(* IEC 61131-3 sources: SmartHomeNew/ (part 17) *)

(* ---- PRG_Telemetry_Causality_Governor.st ---- *)
PROGRAM PRG_Telemetry_Causality_Governor
VAR
    L_Now_MS : UDINT;
    L_Causality_Valid : BOOL := TRUE;
    L_Error_Code : UDINT := 0;
    L_Error_Text : STRING(160) := '';
    L_Ack_Age_MS : UDINT;
    L_Convergence_Age_MS : UDINT;
    L_Stable_Dwell_MS : UDINT;
END_VAR

L_Now_MS := GVL_STATUS.G_System_Time_MS;
L_Causality_Valid := TRUE;
L_Error_Code := 0;
L_Error_Text := '';

// Fail-safe defaults.
GVL_TELEMETRY.Telemetry_Runtime_Valid := FALSE;
GVL_TELEMETRY.Telemetry_Freshness_Valid := FALSE;
GVL_TELEMETRY.Command_Telemetry_Causality_Valid := FALSE;
GVL_TELEMETRY.Actuator_Feedback_Valid := FALSE;
GVL_TELEMETRY.Actuator_Feedback_Fresh := FALSE;
GVL_TELEMETRY.Physical_Effect_Confirmed := FALSE;
GVL_TELEMETRY.Physical_Effect_Finalized := FALSE;
GVL_TELEMETRY.Physical_Target_Converged := FALSE;
GVL_TELEMETRY.Physical_Stable_Window_OK := FALSE;
GVL_TELEMETRY.Command_Telemetry_Divergence_Detected := TRUE;

GVL_TELEMETRY.Command_Epoch := GVL_OUTPUT_EPOCH.Output_Publication_Epoch;

IF NOT GVL_OUTPUT_EPOCH.Output_Publication_Valid THEN
    L_Causality_Valid := FALSE;
    L_Error_Code := 21000;
    L_Error_Text := 'Telemetry causality output publication invalid';
END_IF;

IF L_Causality_Valid AND NOT GVL_OUTPUT_EPOCH.Output_Runtime_Epoch_Valid THEN
    L_Causality_Valid := FALSE;
    L_Error_Code := 21001;
    L_Error_Text := 'Telemetry causality runtime epoch invalid';
END_IF;

IF L_Causality_Valid AND GVL_OUTPUT_EPOCH.Output_Lease_Expired THEN
    L_Causality_Valid := FALSE;
    L_Error_Code := 21002;
    L_Error_Text := 'Telemetry causality output lease expired';
END_IF;

IF L_Causality_Valid AND GVL_OUTPUT_EPOCH.Output_Forced_Safe_Decay THEN
    L_Causality_Valid := FALSE;
    L_Error_Code := 21003;
    L_Error_Text := 'Telemetry causality output forced safe decay';
END_IF;

IF L_Causality_Valid AND (GVL_TELEMETRY.Telemetry_Epoch <> GVL_TELEMETRY.Command_Epoch) THEN
    L_Causality_Valid := FALSE;
    L_Error_Code := 21010;
    L_Error_Text := 'Telemetry epoch does not match command epoch';
END_IF;

IF L_Causality_Valid AND (GVL_TELEMETRY.Telemetry_Epoch < GVL_TELEMETRY.Last_Acknowledged_Command_Epoch) THEN
    GVL_TELEMETRY.Telemetry_Replay_Suspected := TRUE;

    L_Causality_Valid := FALSE;
    L_Error_Code := 21011;
    L_Error_Text := 'Telemetry epoch replay suspected';
END_IF;

L_Ack_Age_MS := L_Now_MS - GVL_TELEMETRY.Last_Physical_Ack_Time_MS;

IF L_Causality_Valid AND (L_Ack_Age_MS > 5000) THEN
    L_Causality_Valid := FALSE;
    L_Error_Code := 21020;
    L_Error_Text := 'Physical acknowledgement stale';
END_IF;

L_Convergence_Age_MS := L_Now_MS - GVL_TELEMETRY.Last_Physical_Convergence_MS;

IF L_Causality_Valid AND (L_Convergence_Age_MS > 10000) THEN
    L_Causality_Valid := FALSE;
    L_Error_Code := 21021;
    L_Error_Text := 'Physical convergence stale';
END_IF;

// Stable physical dwell window.
L_Stable_Dwell_MS :=
    L_Now_MS - GVL_TELEMETRY.Last_Physical_Convergence_MS;

IF L_Causality_Valid AND (L_Stable_Dwell_MS < 3000) THEN
    L_Causality_Valid := FALSE;
    L_Error_Code := 21030;
    L_Error_Text := 'Physical stabilization dwell window incomplete';
END_IF;

// Physical oscillation quarantine.
IF L_Causality_Valid
AND GVL_TELEMETRY.Physical_Oscillation_Detected THEN
    L_Causality_Valid := FALSE;
    L_Error_Code := 21031;
    L_Error_Text := 'Physical oscillation detected';
END_IF;

IF L_Causality_Valid
AND GVL_TELEMETRY.Physical_Transition_Active THEN
    L_Causality_Valid := FALSE;
    L_Error_Code := 21032;
    L_Error_Text := 'Physical transition still active';
END_IF;

IF L_Causality_Valid
AND GVL_TELEMETRY.Physical_Convergence_Replay_Suspected THEN
    L_Causality_Valid := FALSE;
    L_Error_Code := 21033;
    L_Error_Text := 'Physical convergence replay suspected';
END_IF;

IF L_Causality_Valid THEN
    GVL_TELEMETRY.Telemetry_Runtime_Valid := TRUE;
    GVL_TELEMETRY.Telemetry_Freshness_Valid := TRUE;
    GVL_TELEMETRY.Telemetry_Lease_Expired := FALSE;
    GVL_TELEMETRY.Telemetry_Quarantine_Active := FALSE;

    GVL_TELEMETRY.Command_Telemetry_Causality_Valid := TRUE;
    GVL_TELEMETRY.Command_Telemetry_Divergence_Detected := FALSE;

    GVL_TELEMETRY.Actuator_Feedback_Valid := TRUE;
    GVL_TELEMETRY.Actuator_Feedback_Fresh := TRUE;
    GVL_TELEMETRY.Physical_Effect_Confirmed := TRUE;

    GVL_TELEMETRY.Physical_Target_Converged := TRUE;
    GVL_TELEMETRY.Physical_Stable_Window_OK := TRUE;
    GVL_TELEMETRY.Physical_Effect_Finalized := TRUE;

    GVL_TELEMETRY.Last_Acknowledged_Command_Epoch := GVL_TELEMETRY.Command_Epoch;

    GVL_TELEMETRY.Telemetry_Last_Error_Code := 0;
    GVL_TELEMETRY.Telemetry_Last_Error_Text := '';
ELSE
    GVL_TELEMETRY.Telemetry_Runtime_Valid := FALSE;
    GVL_TELEMETRY.Telemetry_Freshness_Valid := FALSE;
    GVL_TELEMETRY.Telemetry_Lease_Expired := TRUE;
    GVL_TELEMETRY.Telemetry_Quarantine_Active := TRUE;

    GVL_TELEMETRY.Command_Telemetry_Causality_Valid := FALSE;
    GVL_TELEMETRY.Command_Telemetry_Divergence_Detected := TRUE;

    GVL_TELEMETRY.Telemetry_Last_Error_Code := L_Error_Code;
    GVL_TELEMETRY.Telemetry_Last_Error_Text := L_Error_Text;
    GVL_TELEMETRY.Telemetry_Invalidation_Count :=
        GVL_TELEMETRY.Telemetry_Invalidation_Count + 1;
END_IF;

END_PROGRAM

(* ---- PRG_Temporal_Domain.st ---- *)
PROGRAM PRG_Temporal_Domain
// SEMANTIC DOMAIN WRAPPER
// PRESERVES ORIGINAL EXECUTION ORDER

PRG_Temporal_Stability_Governor();
PRG_Control_Temporal_Coherence_Governor();

PRG_Temporal_Causality_Closure_Governor();
PRG_Distributed_Epoch_Linearity_Governor();
PRG_Historical_Ordering_Integrity_Governor();
PRG_Causality_Reversal_Prevention_Governor();

END_PROGRAM

(* ---- PRG_Test.st ---- *)
PROGRAM PRG_Test
VAR
    // Инстансы тестируемых блоков
    fbAnalogValidator : FB_Analog_Validator;
    fbRandomGenerator : FB_Random_Generator;
    fbTwoFactorAuth   : FB_TwoFactor_Auth;

    // Переменные для тестов
    L_Test_Step : INT := 0;
    L_Tests_Passed : INT := 0;
    L_Tests_Failed : INT := 0;
    L_System_Time : UDINT := 0;

    // Результаты тестов
    L_Test1_Passed : BOOL;
    L_Test2_Passed : BOOL;
    L_Test3_Passed : BOOL;
END_VAR

// Имитация системного времени
L_System_Time := L_System_Time + 10;

CASE L_Test_Step OF
    0: // Инициализация
        L_Test_Step := 1;

    1: // Тест 1: FB_Analog_Validator - Нормальное значение
        fbAnalogValidator(
            VI_Value := 25.0,
            VI_Min_Valid := 0.0,
            VI_Max_Valid := 50.0,
            VI_Fallback_Mode := 0,
            VI_Default_Value := 20.0
        );
        IF fbAnalogValidator.VO_Valid AND fbAnalogValidator.VO_Validated_Value = 25.0 THEN
            L_Test1_Passed := TRUE;
            L_Tests_Passed := L_Tests_Passed + 1;
        ELSE
            L_Test1_Passed := FALSE;
            L_Tests_Failed := L_Tests_Failed + 1;
        END_IF;
        L_Test_Step := 2;

    2: // Тест 2: FB_Analog_Validator - Выход за границы (Fallback = Default)
        fbAnalogValidator(
            VI_Value := 100.0,
            VI_Min_Valid := 0.0,
            VI_Max_Valid := 50.0,
            VI_Fallback_Mode := 1,
            VI_Default_Value := 20.0
        );
        IF NOT fbAnalogValidator.VO_Valid AND fbAnalogValidator.VO_Validated_Value = 20.0 THEN
            L_Test2_Passed := TRUE;
            L_Tests_Passed := L_Tests_Passed + 1;
        ELSE
            L_Test2_Passed := FALSE;
            L_Tests_Failed := L_Tests_Failed + 1;
        END_IF;
        L_Test_Step := 3;

    3: // Тест 3: FB_Random_Generator - Диапазон
        fbRandomGenerator.Seed(12345);
        fbRandomGenerator.Random_Int_Range(VI_min := 10, VI_max := 20, VI_System_Time_MS := L_System_Time);
        IF fbRandomGenerator.VO_Random_Value >= 10 AND fbRandomGenerator.VO_Random_Value <= 20 THEN
            L_Test3_Passed := TRUE;
            L_Tests_Passed := L_Tests_Passed + 1;
        ELSE
            L_Test3_Passed := FALSE;
            L_Tests_Failed := L_Tests_Failed + 1;
        END_IF;
        L_Test_Step := 100; // Завершение тестов

    100: // Тесты завершены
        // Здесь можно вывести результаты в лог или HMI
        ;
END_CASE;
// >>> BULK_SYNC_ANCHOR: PRG_Test <<<

(* ---- PRG_Test_Scenario_Runner.st ---- *)
PROGRAM PRG_Test_Scenario_Runner

IF NOT GVL_TEST.G_Test_Enable THEN
    RETURN;
END_IF;

CASE GVL_TEST_INJECTION.G_Test_Step OF

0:
    // idle

1:
    // simulate gas spike
    GVL_TEST_INJECTION.G_Inject_Gas_Level := 50.0;
    GVL_TEST_INJECTION.G_Test_Step := 2;

2:
    // simulate illegal reset
    GVL_TEST_INJECTION.G_Inject_Force_Gas_Alarm_Reset := TRUE;
    GVL_TEST_INJECTION.G_Test_Step := 3;

3:
    // simulate IO offline
    GVL_TEST_INJECTION.G_Inject_Force_IO_Offline := TRUE;
    GVL_TEST_INJECTION.G_Test_Step := 4;

4:
    // stop
    GVL_TEST_INJECTION.G_Inject_Enable := FALSE;

END_CASE;

(* ---- PRG_Time_Service.st ---- *)
PROGRAM PRG_Time_Service
VAR
    fbTimebase : FB_System_Timebase;
    fbTime : FB_Time_Service;
END_VAR

// Central time update point.
// Must run before PRG_IO_Read and all consumers of GVL_TIME_SERVICE.
fbTimebase();
fbTime();

// Step 4.2 compatibility bridge.
// Legacy consumers of GVL_STATUS.G_System_Time_MS receive the same canonical time.
GVL_STATUS.G_System_Time_MS := GVL_TIME_SERVICE.G_Now_MS;
GVL_STATUS.G_Current_TOD := GVL_TIME_SERVICE.G_Current_TOD;
GVL_STATUS.G_Current_Day := GVL_TIME_SERVICE.G_Day_Of_Week;

END_PROGRAM

(* ---- PRG_Transport_Freshness_Governor.st ---- *)
PROGRAM PRG_Transport_Freshness_Governor
VAR
    L_Now_MS : UDINT;
    L_Delta_MS : UDINT;
    L_Transport_Valid : BOOL := TRUE;
    L_Error_Code : UDINT := 0;
    L_Error_Text : STRING(160) := '';
END_VAR

L_Now_MS := GVL_STATUS.G_System_Time_MS;
L_Transport_Valid := TRUE;
L_Error_Code := 0;
L_Error_Text := '';

// ======================================================
// TRANSPORT FRESHNESS GOVERNOR
// ======================================================
// Governs transport freshness semantics.
// Prevents stale transport semantic publication.
// ======================================================

GVL_TRANSPORT_FRESHNESS.Transport_Stale_Frame_Detected := FALSE;
GVL_TRANSPORT_FRESHNESS.Transport_Transaction_Mismatch := FALSE;
GVL_TRANSPORT_FRESHNESS.Transport_Snapshot_Invalid := FALSE;

// Runtime authority linkage.
IF NOT GVL_RUNTIME_EPOCH.Runtime_Runtime_Barrier_OK THEN
    L_Transport_Valid := FALSE;
    L_Error_Code := 10000;
    L_Error_Text := 'Transport runtime authority invalid';
END_IF;

// Monotonic authority linkage.
IF L_Transport_Valid AND (NOT GVL_TIME_MONOTONIC.Monotonic_Time_Valid) THEN
    L_Transport_Valid := FALSE;
    L_Error_Code := 10001;
    L_Error_Text := 'Transport monotonic authority invalid';
END_IF;

// Recovery governance linkage.
IF L_Transport_Valid AND GVL_RECOVERY_GOVERNANCE.Recovery_Quarantine_Active THEN
    L_Transport_Valid := FALSE;
    L_Error_Code := 10002;
    L_Error_Text := 'Transport blocked by recovery quarantine';
END_IF;

// Transport reconnect quarantine.
IF GVL_TRANSPORT_FRESHNESS.Transport_Reconnect_Stabilizing THEN
    GVL_TRANSPORT_FRESHNESS.Transport_Quarantine_Active := TRUE;

    L_Transport_Valid := FALSE;

    IF L_Error_Code = 0 THEN
        L_Error_Code := 10003;
        L_Error_Text := 'Transport reconnect stabilization active';
    END_IF;
END_IF;

// Lease freshness validation.
L_Delta_MS := L_Now_MS - GVL_TRANSPORT_FRESHNESS.Transport_Last_Refresh_MS;

IF L_Transport_Valid AND GVL_TRANSPORT_FRESHNESS.Transport_Lease_Valid THEN
    IF L_Delta_MS > GVL_TRANSPORT_FRESHNESS.Transport_Lease_Timeout_MS THEN
        L_Transport_Valid := FALSE;
        L_Error_Code := 10004;
        L_Error_Text := 'Transport lease expired';

        GVL_TRANSPORT_FRESHNESS.Transport_Lease_Expired := TRUE;
    END_IF;
END_IF;

// Publish authoritative transport freshness state.
IF L_Transport_Valid THEN
    GVL_TRANSPORT_FRESHNESS.Transport_Epoch := GVL_TRANSPORT_FRESHNESS.Transport_Epoch + 1;
    GVL_TRANSPORT_FRESHNESS.Transport_Publication_Epoch := GVL_TRANSPORT_FRESHNESS.Transport_Publication_Epoch + 1;

    GVL_TRANSPORT_FRESHNESS.Transport_Freshness_Valid := TRUE;
    GVL_TRANSPORT_FRESHNESS.Transport_Publication_Allowed := TRUE;

    GVL_TRANSPORT_FRESHNESS.Transport_Lease_Valid := TRUE;
    GVL_TRANSPORT_FRESHNESS.Transport_Lease_Expired := FALSE;

    GVL_TRANSPORT_FRESHNESS.Transport_Quarantine_Active := FALSE;

    GVL_TRANSPORT_FRESHNESS.Transport_Last_Refresh_MS := L_Now_MS;
    GVL_TRANSPORT_FRESHNESS.Transport_Last_Publication_MS := L_Now_MS;

    GVL_TRANSPORT_FRESHNESS.Transport_Last_Error_Code := 0;
    GVL_TRANSPORT_FRESHNESS.Transport_Last_Error_Text := '';
ELSE
    GVL_TRANSPORT_FRESHNESS.Transport_Freshness_Valid := FALSE;
    GVL_TRANSPORT_FRESHNESS.Transport_Publication_Allowed := FALSE;

    GVL_TRANSPORT_FRESHNESS.Transport_Snapshot_Invalid := TRUE;

    GVL_TRANSPORT_FRESHNESS.Transport_Last_Error_Code := L_Error_Code;
    GVL_TRANSPORT_FRESHNESS.Transport_Last_Error_Text := L_Error_Text;

    GVL_TRANSPORT_FRESHNESS.Transport_Invalidation_Count := GVL_TRANSPORT_FRESHNESS.Transport_Invalidation_Count + 1;
END_IF;
END_PROGRAM

(* ---- PRG_Unsafe_Transition_Forensics_Governor.st ---- *)
PROGRAM PRG_Unsafe_Transition_Forensics_Governor
IF GVL_PHYSICAL_SAFETY_PROJECTION_FABRIC.Physical_Safety_Projection_Granted
AND NOT GVL_UNSAFE_TRANSITION_FORENSICS_FABRIC.Unsafe_Transition_Hidden
AND NOT GVL_UNSAFE_TRANSITION_FORENSICS_FABRIC.Forensic_Lineage_Break_Detected
AND NOT GVL_UNSAFE_TRANSITION_FORENSICS_FABRIC.Historical_Safety_Gap_Detected THEN

    GVL_UNSAFE_TRANSITION_FORENSICS_FABRIC.Unsafe_Transition_Forensics_Valid := TRUE;
    GVL_UNSAFE_TRANSITION_FORENSICS_FABRIC.Unsafe_Transition_Forensics_Granted := TRUE;
    GVL_UNSAFE_TRANSITION_FORENSICS_FABRIC.Unsafe_Transition_Lineage_Preserved := TRUE;
    GVL_UNSAFE_TRANSITION_FORENSICS_FABRIC.Forensic_Causality_Continuity_Valid := TRUE;
    GVL_UNSAFE_TRANSITION_FORENSICS_FABRIC.Distributed_Unsafe_Event_Consensus := TRUE;
END_IF;
END_PROGRAM

(* ---- PRG_User_Adapt_Control.st ---- *)
PROGRAM PRG_User_Adapt_Control
VAR
    fbTrace : FB_Trace_Write;
    L_Text : STRING(64);
END_VAR

IF GVL_INTENT_USER.I_Set_Adapt_Profile_Req THEN

    // block if safety active
    IF (GVL_SAFETY_SHUTDOWN.G_Safety_Mode <> NORMAL) OR GVL_SAFETY_RECOVERY.G_Recovery_Active THEN

        fbTrace(
            iLayer := TRACE_USER,
            iSource := SRC_USER,
            iReason := REASON_SAFETY,
            iValueBool := FALSE,
            iValueReal := 0.0,
            iText := 'Profile change blocked: SAFETY ACTIVE'
        );

    ELSE

        IF (GVL_INTENT_USER.I_Set_Adapt_Profile_Confirm)
           AND (GVL_INTENT_USER.I_User_Access_Level >= 2) THEN

            GVL_BEHAVIOR_ADAPT.G_Adapt_Profile :=
                GVL_INTENT_USER.I_Adapt_Profile_Value;

            IF GVL_INTENT_USER.I_Adapt_Profile_Value = ADAPT_PROFILE_STABLE THEN
                L_Text := 'Adapt profile: STABLE';
            ELSIF GVL_INTENT_USER.I_Adapt_Profile_Value = ADAPT_PROFILE_BALANCED THEN
                L_Text := 'Adapt profile: BALANCED';
            ELSE
                L_Text := 'Adapt profile: AGGRESSIVE';
            END_IF;

            fbTrace(
                iLayer := TRACE_USER,
                iSource := SRC_USER,
                iReason := REASON_USER_REQUEST,
                iValueBool := TRUE,
                iValueReal := TO_REAL(GVL_INTENT_USER.I_User_Access_Level),
                iText := L_Text
            );

        END_IF;

    END_IF;

    GVL_INTENT_USER.I_Set_Adapt_Profile_Req := FALSE;
    GVL_INTENT_USER.I_Set_Adapt_Profile_Confirm := FALSE;

END_IF;

(* ---- PRG_Ventilation.st ---- *)
PROGRAM PRG_Ventilation
VAR
    fbVentilationManager : FB_Ventilation_System_Manager;
    fbVentProjection : FB_Vent_Output_Projection;

    L_i : INT;

    L_Supply_Fans_Byte : ARRAY[1..GVL_CONSTANTS.C_MAX_SUPPLY_FANS] OF BYTE;
    L_Exhaust_Fans_Byte : ARRAY[1..GVL_CONSTANTS.C_MAX_EXHAUST_FANS] OF BYTE;

    L_Wet_Zone_Active : ARRAY[1..GVL_CONSTANTS.C_MAX_WET_ZONES] OF BOOL;

    L_Vent_PV3_Boost_Req : BOOL;
    L_Supply_100_Req : BOOL;
    L_Exhaust_100_Req : BOOL;
    L_Supply_80_Req : BOOL;
    L_Vent_Stop_Req : BOOL;

    L_Distributed_Execute_Allowed : BOOL;
    L_Distributed_Projection_Allowed : BOOL;

    L_Fire_Smoke_Override : BOOL;
    L_Gas_Vent_Override : BOOL;
    L_Safety_Vent_Override : BOOL;
END_VAR

FOR L_i := 1 TO GVL_CONSTANTS.C_MAX_SUPPLY_FANS DO
    L_Supply_Fans_Byte[L_i] := 0;
END_FOR;

FOR L_i := 1 TO GVL_CONSTANTS.C_MAX_EXHAUST_FANS DO
    L_Exhaust_Fans_Byte[L_i] := 0;
END_FOR;

L_Distributed_Execute_Allowed :=
    GVL_Distributed_Execution_Gates.G_Can_Execute;

L_Distributed_Projection_Allowed :=
    GVL_Distributed_Execution_Gates.G_Can_Own_Projection;

L_Fire_Smoke_Override :=
    GVL_COMMAND_SHADOW.G_Vent_Smoke_Exhaust;

L_Gas_Vent_Override :=
    (GVL_SAFETY_SHUTDOWN.G_Safety_Mode = GAS)
    OR GVL_COMMAND_SHADOW.G_Vent_PV3_Boost
    OR GVL_COMMAND_SHADOW.G_Supply_100_Req;

L_Vent_PV3_Boost_Req := GVL_COMMAND_SHADOW.G_Vent_PV3_Boost;
L_Supply_100_Req := GVL_COMMAND_SHADOW.G_Supply_100_Req;
L_Exhaust_100_Req := GVL_COMMAND_SHADOW.G_Exhaust_100_Req;
L_Supply_80_Req := GVL_COMMAND_SHADOW.G_Supply_80_Req;
L_Vent_Stop_Req := GVL_COMMAND_SHADOW.G_Vent_Stop;

L_Safety_Vent_Override :=
    L_Fire_Smoke_Override
    OR L_Gas_Vent_Override
    OR L_Supply_80_Req
    OR L_Exhaust_100_Req;

FOR L_i := 1 TO GVL_CONSTANTS.C_MAX_WET_ZONES DO
    L_Wet_Zone_Active[L_i] := FALSE;
END_FOR;

IF GVL_STATUS.G_Wet_Zone_Light_Active THEN
    L_Wet_Zone_Active[1] := TRUE;
END_IF;

IF L_Distributed_Execute_Allowed THEN
    fbVentilationManager(
        VI_System_Time_MS := GVL_STATUS.G_System_Time_MS,
        VI_IsActivePLC := GVL_STATUS.G_Is_Active_PLC,
        VI_Outdoor_Temp := GVL_STATE.G_Outdoor_Temp,
        VI_Supply_Temps := GVL_STATE.G_Supply_Temps,
        VI_Room_Temps := GVL_STATE.G_Room_Temps,
        VI_Room_Humidities := GVL_STATE.G_Room_Hum,
        VI_Room_CO2 := GVL_STATE.G_Room_CO2,
        VI_Current_Scenario := GVL_STATUS.G_Current_Scenario,
        VI_System_Mode := GVL_STATE.G_System_Mode,
        VI_Config := GVL_CONFIG.G_HMI_Vent_Global_Config,
        VI_Fire_Alarm := GVL_STATE.G_Safety_Smoke_Latched,
        VI_Gas_Alarm := GVL_STATE.G_Safety_Gas_Latched,
        VI_PV3_Boost_Req := L_Vent_PV3_Boost_Req,
        VI_Supply_100_Req := L_Supply_100_Req,
        VI_Exhaust_100_Req := L_Exhaust_100_Req,
        VI_Supply_80_Req := L_Supply_80_Req,
        VI_Vent_Stop := L_Vent_Stop_Req,
        VI_IO_Modules_Online := GVL_STATUS.G_IO_Modules_Online,
        VI_Wet_Zone_Active := L_Wet_Zone_Active,
        VI_Rule_Actions := GVL_STATE.G_Rule_Actions,
        VO_Supply_Fans => L_Supply_Fans_Byte,
        VO_Exhaust_Fans => L_Exhaust_Fans_Byte,
        VO_Heater_Power => GVL_STATE.G_Vent_Heater_Power,
        VO_Status_Msg => GVL_STATUS.G_Vent_Status_Msg,
        VO_Ventilation_IO_Fault => GVL_STATE.G_Ventilation_IO_Fault,
        VO_Ventilation_Subsystem_Degraded => GVL_STATE.G_Ventilation_Subsystem_Degraded
    );
END_IF;

IF L_Fire_Smoke_Override THEN
    FOR L_i := 1 TO GVL_CONSTANTS.C_MAX_EXHAUST_FANS DO
        L_Exhaust_Fans_Byte[L_i] := 100;
    END_FOR;

    FOR L_i := 1 TO GVL_CONSTANTS.C_MAX_SUPPLY_FANS DO
        L_Supply_Fans_Byte[L_i] := 0;
    END_FOR;
ELSIF L_Supply_100_Req THEN
    FOR L_i := 1 TO GVL_CONSTANTS.C_MAX_SUPPLY_FANS DO
        L_Supply_Fans_Byte[L_i] := 100;
    END_FOR;
ELSIF L_Supply_80_Req THEN
    FOR L_i := 1 TO GVL_CONSTANTS.C_MAX_SUPPLY_FANS DO
        IF L_Supply_Fans_Byte[L_i] < 80 THEN
            L_Supply_Fans_Byte[L_i] := 80;
        END_IF;
    END_FOR;
END_IF;

IF (NOT L_Fire_Smoke_Override) AND L_Vent_PV3_Boost_Req THEN
    IF GVL_CONSTANTS.C_MAX_SUPPLY_FANS >= 3 THEN
        L_Supply_Fans_Byte[3] := 100;
    ELSE
        L_Supply_Fans_Byte[1] := 100;
    END_IF;
END_IF;

IF (NOT L_Fire_Smoke_Override) AND L_Exhaust_100_Req THEN
    FOR L_i := 1 TO GVL_CONSTANTS.C_MAX_EXHAUST_FANS DO
        L_Exhaust_Fans_Byte[L_i] := 100;
    END_FOR;
END_IF;

IF L_Vent_Stop_Req AND NOT L_Safety_Vent_Override THEN
    FOR L_i := 1 TO GVL_CONSTANTS.C_MAX_SUPPLY_FANS DO
        L_Supply_Fans_Byte[L_i] := 0;
    END_FOR;
    FOR L_i := 1 TO GVL_CONSTANTS.C_MAX_EXHAUST_FANS DO
        L_Exhaust_Fans_Byte[L_i] := 0;
    END_FOR;
END_IF;

IF NOT L_Distributed_Projection_Allowed
   AND NOT L_Safety_Vent_Override THEN

    FOR L_i := 1 TO GVL_CONSTANTS.C_MAX_EXHAUST_FANS DO
        L_Exhaust_Fans_Byte[L_i] := 0;
    END_FOR;

    FOR L_i := 1 TO GVL_CONSTANTS.C_MAX_SUPPLY_FANS DO
        L_Supply_Fans_Byte[L_i] := 0;
    END_FOR;
END_IF;

fbVentProjection(
    VI_Supply_Fans := L_Supply_Fans_Byte,
    VI_Exhaust_Fans := L_Exhaust_Fans_Byte
);

// >>> BULK_SYNC_ANCHOR: PRG_Ventilation <<<
END_PROGRAM

(* ---- PRG_Verification_Domain.st ---- *)
PROGRAM PRG_Verification_Domain
// SEMANTIC DOMAIN WRAPPER

PRG_Passive_Runtime_Verification_Governor();
PRG_Semantic_Drift_Observability_Governor();
PRG_Proof_Continuity_Audit_Governor();
PRG_Runtime_Assumption_Integrity_Governor();

PRG_Command_Verifier();
PRG_Explainability();

END_PROGRAM

(* ---- PRG_Water.st ---- *)
PROGRAM PRG_Water
VAR
    fbProjection : FB_Water_Output_Projection;
    L_Zone_Enable : ARRAY[1..GVL_CONSTANTS.C_MAX_WATER_ZONES] OF BOOL;
    L_Valve_35_Close : BOOL;
    L_Valve_36_Close : BOOL;
    L_i : INT;
    L_Projected_Valve_Group : UINT;
END_VAR

// ==============================================================================
// Water runtime output bridge.
//
// GVL_COMMAND_SHADOW remains owned exclusively by PRG_Command_Arbitration.
// This PRG is the water domain output projection bridge into GVL_WATER_OUTPUT.
//
// Normally-open water valves policy:
// - normal state is open;
// - leak/fallback projects close command;
// - HMI emergency-open is a timed, limited suppression of the close command,
//   not a direct physical-output write.
// ==============================================================================

PRG_Water_Emergency_Open_Manager();

GVL_WATER_DOMAIN_STATUS.G_Runtime_Required := FALSE;
GVL_WATER_DOMAIN_STATUS.G_Runtime_Executed := TRUE;
GVL_WATER_DOMAIN_STATUS.G_Runtime_Idle_By_Design := FALSE;
GVL_WATER_DOMAIN_STATUS.G_Recovery_Requested := FALSE;
GVL_WATER_DOMAIN_STATUS.G_Global_Path_Active := FALSE;
GVL_WATER_DOMAIN_STATUS.G_Output_35_Active := FALSE;
GVL_WATER_DOMAIN_STATUS.G_Output_36_Active := FALSE;
GVL_WATER_DOMAIN_STATUS.G_Any_Zone_Active := FALSE;
GVL_WATER_DOMAIN_STATUS.G_Last_Update_MS := GVL_STATUS.G_System_Time_MS;

FOR L_i := 1 TO GVL_CONSTANTS.C_MAX_WATER_ZONES DO
    L_Zone_Enable[L_i] := FALSE;
END_FOR;

IF GVL_INTENT_SAFETY.I_Water_Selective_Recovery_Allowed THEN
    GVL_WATER_DOMAIN_STATUS.G_Recovery_Requested := TRUE;

    IF (GVL_INTENT_SAFETY.I_Water_Recovery_Target_Zone >= 1) AND (GVL_INTENT_SAFETY.I_Water_Recovery_Target_Zone <= GVL_CONSTANTS.C_MAX_WATER_ZONES) THEN
        L_Zone_Enable[GVL_INTENT_SAFETY.I_Water_Recovery_Target_Zone] := TRUE;
    END_IF;
END_IF;

// Existing authoritative global fallback path.
L_Valve_35_Close := GVL_COMMAND_SHADOW.G_Close_Valve_35;
L_Valve_36_Close := GVL_COMMAND_SHADOW.G_Close_Valve_36;

// Deterministic projection bridge.
// Conservative global fallback projection dominates selective projection.
IF GVL_Water_Output_Projection.G_Runtime_Valid THEN

    IF GVL_Water_Output_Projection.G_Global_Fallback_Projecting THEN
        L_Valve_35_Close := TRUE;
        L_Valve_36_Close := TRUE;
        GVL_WATER_DOMAIN_STATUS.G_Global_Path_Active := TRUE;
    ELSE
        FOR L_i := 1 TO GVL_CONSTANTS.C_MAX_FLOOD_SENSORS DO
            IF GVL_Water_Output_Projection.G_Output_Projection_State[L_i].Projection_Allowed AND
               GVL_Water_Output_Projection.G_Output_Projection_State[L_i].Physical_Close_Project THEN

                L_Projected_Valve_Group :=
                    GVL_Water_Output_Projection.G_Output_Projection_State[L_i].Valve_Group_Id;

                CASE L_Projected_Valve_Group OF
                    1:
                        L_Valve_35_Close := TRUE;
                    2:
                        L_Valve_36_Close := TRUE;
                    3:
                        L_Valve_35_Close := TRUE;
                        L_Valve_36_Close := TRUE;
                ELSE
                    // Unknown valve group is not projected here.
                    // Conservative fallback is handled by authority/projection layers.
                END_CASE;
            END_IF;
        END_FOR;
    END_IF;
END_IF;

// Emergency open for normally-open valves: temporarily remove close projection.
IF GVL_WATER_EMERGENCY_OPEN.G_Open_Valve_35_Active THEN
    L_Valve_35_Close := FALSE;
END_IF;

IF GVL_WATER_EMERGENCY_OPEN.G_Open_Valve_36_Active THEN
    L_Valve_36_Close := FALSE;
END_IF;

FOR L_i := 1 TO GVL_CONSTANTS.C_MAX_WATER_ZONES DO
    IF L_Zone_Enable[L_i] THEN
        GVL_WATER_DOMAIN_STATUS.G_Any_Zone_Active := TRUE;
    END_IF;
END_FOR;

GVL_WATER_DOMAIN_STATUS.G_Output_35_Active := L_Valve_35_Close;
GVL_WATER_DOMAIN_STATUS.G_Output_36_Active := L_Valve_36_Close;

GVL_WATER_DOMAIN_STATUS.G_Runtime_Required :=
    GVL_WATER_DOMAIN_STATUS.G_Recovery_Requested
    OR GVL_WATER_DOMAIN_STATUS.G_Global_Path_Active
    OR GVL_WATER_DOMAIN_STATUS.G_Output_35_Active
    OR GVL_WATER_DOMAIN_STATUS.G_Output_36_Active
    OR GVL_WATER_DOMAIN_STATUS.G_Any_Zone_Active;

GVL_WATER_DOMAIN_STATUS.G_Runtime_Idle_By_Design :=
    NOT GVL_WATER_DOMAIN_STATUS.G_Runtime_Required;

IF GVL_WATER_DOMAIN_STATUS.G_Runtime_Idle_By_Design THEN
    GVL_WATER_DOMAIN_STATUS.G_Status_Code := 0;
    GVL_WATER_DOMAIN_STATUS.G_Status_Text := 'Water domain idle by design';
ELSIF GVL_WATER_DOMAIN_STATUS.G_Global_Path_Active THEN
    GVL_WATER_DOMAIN_STATUS.G_Status_Code := 2;
    GVL_WATER_DOMAIN_STATUS.G_Status_Text := 'Water domain global path active';
ELSIF GVL_WATER_EMERGENCY_OPEN.G_Open_Valve_35_Active OR GVL_WATER_EMERGENCY_OPEN.G_Open_Valve_36_Active THEN
    GVL_WATER_DOMAIN_STATUS.G_Status_Code := 3;
    GVL_WATER_DOMAIN_STATUS.G_Status_Text := 'Water emergency open active';
ELSE
    GVL_WATER_DOMAIN_STATUS.G_Status_Code := 1;
    GVL_WATER_DOMAIN_STATUS.G_Status_Text := 'Water domain active';
END_IF;

fbProjection(
    VI_Zone_Enable := L_Zone_Enable,
    VI_Valve_35_Close := L_Valve_35_Close,
    VI_Valve_36_Close := L_Valve_36_Close
);

// >>> BULK_SYNC_ANCHOR: PRG_Water <<<
END_PROGRAM

(* ---- PRG_Water_Emergency_Open_Manager.st ---- *)
PROGRAM PRG_Water_Emergency_Open_Manager
VAR
    L_Group : INT;
    L_Duration_MS : UDINT;
    L_Elapsed_MS : UDINT;
    L_Remaining_MS : UDINT;
    L_Leak_Active : BOOL;
    L_i : INT;
END_VAR

// Daily limit reset on monotonic 24h window.
IF (GVL_WATER_EMERGENCY_OPEN.G_Daily_Reset_MS = 0) OR
   ((GVL_TIME_SERVICE.G_Now_MS - GVL_WATER_EMERGENCY_OPEN.G_Daily_Reset_MS) >= GVL_CONSTANTS.C_MS_IN_DAY) THEN
    FOR L_i := 1 TO 4 DO
        GVL_WATER_EMERGENCY_OPEN.G_Open_Count_Today[L_i] := 0;
    END_FOR;
    GVL_WATER_EMERGENCY_OPEN.G_Daily_Reset_MS := GVL_TIME_SERVICE.G_Now_MS;
END_IF;

L_Leak_Active := GVL_STATE.G_Safety_Leak_Alarm OR GVL_STATE.G_Safety_Leak_Latched;

// HMI immediate close before timeout.
IF GVL_WATER_EMERGENCY_OPEN.G_Request_Close_Now THEN
    L_Group := GVL_WATER_EMERGENCY_OPEN.G_Target_Isolation_Group;

    GVL_WATER_EMERGENCY_OPEN.G_Last_Request_Accepted := FALSE;
    GVL_WATER_EMERGENCY_OPEN.G_Last_Request_Denied := FALSE;
    GVL_WATER_EMERGENCY_OPEN.G_Last_Denial_Code := 0;
    GVL_WATER_EMERGENCY_OPEN.G_Last_Event_Group := L_Group;
    GVL_WATER_EMERGENCY_OPEN.G_Last_Event_MS := GVL_TIME_SERVICE.G_Now_MS;

    IF (L_Group >= 1) AND (L_Group <= 4) THEN
        GVL_WATER_EMERGENCY_OPEN.G_Open_Active[L_Group] := FALSE;
        GVL_WATER_EMERGENCY_OPEN.G_Open_Duration_MS[L_Group] := 0;
        GVL_WATER_EMERGENCY_OPEN.G_Open_Remaining_MS[L_Group] := 0;
        GVL_WATER_EMERGENCY_OPEN.G_Status_Text := 'Emergency open cancelled by HMI';
    ELSE
        FOR L_i := 1 TO 4 DO
            GVL_WATER_EMERGENCY_OPEN.G_Open_Active[L_i] := FALSE;
            GVL_WATER_EMERGENCY_OPEN.G_Open_Duration_MS[L_i] := 0;
            GVL_WATER_EMERGENCY_OPEN.G_Open_Remaining_MS[L_i] := 0;
        END_FOR;
        GVL_WATER_EMERGENCY_OPEN.G_Status_Text := 'All emergency opens cancelled by HMI';
    END_IF;

    GVL_WATER_EMERGENCY_OPEN.G_Request_Close_Now := FALSE;
END_IF;

// HMI emergency open request.
// Groups 1..3 = local risers; group 4 = common inlet 35/36.
IF GVL_WATER_EMERGENCY_OPEN.G_Request_Open THEN
    L_Group := GVL_WATER_EMERGENCY_OPEN.G_Target_Isolation_Group;
    L_Duration_MS := 0;

    GVL_WATER_EMERGENCY_OPEN.G_Last_Request_Accepted := FALSE;
    GVL_WATER_EMERGENCY_OPEN.G_Last_Request_Denied := FALSE;
    GVL_WATER_EMERGENCY_OPEN.G_Last_Denial_Code := 0;
    GVL_WATER_EMERGENCY_OPEN.G_Last_Event_Group := L_Group;
    GVL_WATER_EMERGENCY_OPEN.G_Last_Event_MS := GVL_TIME_SERVICE.G_Now_MS;

    CASE GVL_WATER_EMERGENCY_OPEN.G_Duration_Minutes OF
        1:
            L_Duration_MS := GVL_CONSTANTS.C_MS_IN_MINUTE;
        3:
            L_Duration_MS := GVL_CONSTANTS.C_MS_IN_MINUTE * 3;
        5:
            L_Duration_MS := GVL_CONSTANTS.C_MS_IN_MINUTE * 5;
    ELSE
            L_Duration_MS := 0;
    END_CASE;

    IF NOT L_Leak_Active THEN
        GVL_WATER_EMERGENCY_OPEN.G_Last_Request_Denied := TRUE;
        GVL_WATER_EMERGENCY_OPEN.G_Last_Denial_Code := 1;
        GVL_WATER_EMERGENCY_OPEN.G_Status_Text := 'Emergency open denied: no active leak alarm';
    ELSIF GVL_INTENT_USER.I_User_Access_Level < 2 THEN
        GVL_WATER_EMERGENCY_OPEN.G_Last_Request_Denied := TRUE;
        GVL_WATER_EMERGENCY_OPEN.G_Last_Denial_Code := 2;
        GVL_WATER_EMERGENCY_OPEN.G_Status_Text := 'Emergency open denied: access level < 2';
    ELSIF (L_Group < 1) OR (L_Group > 4) THEN
        GVL_WATER_EMERGENCY_OPEN.G_Last_Request_Denied := TRUE;
        GVL_WATER_EMERGENCY_OPEN.G_Last_Denial_Code := 3;
        GVL_WATER_EMERGENCY_OPEN.G_Status_Text := 'Emergency open denied: invalid isolation group';
    ELSIF L_Duration_MS = 0 THEN
        GVL_WATER_EMERGENCY_OPEN.G_Last_Request_Denied := TRUE;
        GVL_WATER_EMERGENCY_OPEN.G_Last_Denial_Code := 4;
        GVL_WATER_EMERGENCY_OPEN.G_Status_Text := 'Emergency open denied: invalid duration';
    ELSIF GVL_WATER_EMERGENCY_OPEN.G_Open_Count_Today[L_Group] >= 3 THEN
        GVL_WATER_EMERGENCY_OPEN.G_Last_Request_Denied := TRUE;
        GVL_WATER_EMERGENCY_OPEN.G_Last_Denial_Code := 5;
        GVL_WATER_EMERGENCY_OPEN.G_Status_Text := 'Emergency open denied: daily limit reached';
    ELSE
        GVL_WATER_EMERGENCY_OPEN.G_Open_Active[L_Group] := TRUE;
        GVL_WATER_EMERGENCY_OPEN.G_Open_Start_MS[L_Group] := GVL_TIME_SERVICE.G_Now_MS;
        GVL_WATER_EMERGENCY_OPEN.G_Open_Duration_MS[L_Group] := L_Duration_MS;
        GVL_WATER_EMERGENCY_OPEN.G_Open_Remaining_MS[L_Group] := L_Duration_MS;
        GVL_WATER_EMERGENCY_OPEN.G_Open_Count_Today[L_Group] := GVL_WATER_EMERGENCY_OPEN.G_Open_Count_Today[L_Group] + 1;
        GVL_WATER_EMERGENCY_OPEN.G_Last_Request_Accepted := TRUE;
        GVL_WATER_EMERGENCY_OPEN.G_Status_Text := 'Emergency open accepted';
    END_IF;

    GVL_WATER_EMERGENCY_OPEN.G_Request_Open := FALSE;
END_IF;

GVL_WATER_EMERGENCY_OPEN.G_Any_Open_Active := FALSE;

// Timeout and remaining-time management.
FOR L_i := 1 TO 4 DO
    IF GVL_WATER_EMERGENCY_OPEN.G_Open_Active[L_i] THEN
        IF GVL_TIME_SERVICE.G_Now_MS >= GVL_WATER_EMERGENCY_OPEN.G_Open_Start_MS[L_i] THEN
            L_Elapsed_MS := GVL_TIME_SERVICE.G_Now_MS - GVL_WATER_EMERGENCY_OPEN.G_Open_Start_MS[L_i];
        ELSE
            L_Elapsed_MS := (4294967295 - GVL_WATER_EMERGENCY_OPEN.G_Open_Start_MS[L_i]) + GVL_TIME_SERVICE.G_Now_MS + 1;
        END_IF;

        IF L_Elapsed_MS >= GVL_WATER_EMERGENCY_OPEN.G_Open_Duration_MS[L_i] THEN
            GVL_WATER_EMERGENCY_OPEN.G_Open_Active[L_i] := FALSE;
            GVL_WATER_EMERGENCY_OPEN.G_Open_Duration_MS[L_i] := 0;
            GVL_WATER_EMERGENCY_OPEN.G_Open_Remaining_MS[L_i] := 0;
            GVL_WATER_EMERGENCY_OPEN.G_Last_Event_Group := L_i;
            GVL_WATER_EMERGENCY_OPEN.G_Last_Event_MS := GVL_TIME_SERVICE.G_Now_MS;
            GVL_WATER_EMERGENCY_OPEN.G_Status_Text := 'Emergency open timeout elapsed';
        ELSE
            L_Remaining_MS := GVL_WATER_EMERGENCY_OPEN.G_Open_Duration_MS[L_i] - L_Elapsed_MS;
            GVL_WATER_EMERGENCY_OPEN.G_Open_Remaining_MS[L_i] := L_Remaining_MS;
            GVL_WATER_EMERGENCY_OPEN.G_Any_Open_Active := TRUE;
        END_IF;
    ELSE
        GVL_WATER_EMERGENCY_OPEN.G_Open_Remaining_MS[L_i] := 0;
    END_IF;
END_FOR;

GVL_WATER_EMERGENCY_OPEN.G_Open_Riser_1_Active := GVL_WATER_EMERGENCY_OPEN.G_Open_Active[1];
GVL_WATER_EMERGENCY_OPEN.G_Open_Riser_2_Active := GVL_WATER_EMERGENCY_OPEN.G_Open_Active[2];
GVL_WATER_EMERGENCY_OPEN.G_Open_Riser_3_Active := GVL_WATER_EMERGENCY_OPEN.G_Open_Active[3];
GVL_WATER_EMERGENCY_OPEN.G_Open_Common_Inlet_Active := GVL_WATER_EMERGENCY_OPEN.G_Open_Active[4];
GVL_WATER_EMERGENCY_OPEN.G_Any_Open_Active :=
    GVL_WATER_EMERGENCY_OPEN.G_Open_Riser_1_Active OR
    GVL_WATER_EMERGENCY_OPEN.G_Open_Riser_2_Active OR
    GVL_WATER_EMERGENCY_OPEN.G_Open_Riser_3_Active OR
    GVL_WATER_EMERGENCY_OPEN.G_Open_Common_Inlet_Active;
GVL_WATER_EMERGENCY_OPEN.G_Last_Update_MS := GVL_TIME_SERVICE.G_Now_MS;

END_PROGRAM

(* ---- PRG_Water_Output_Projection.st ---- *)
PROGRAM PRG_Water_Output_Projection
VAR
    fbWaterOutputProjector : FB_Water_Output_Projector;
    fbWaterOutputReconciliation : FB_Water_Output_Reconciliation;
END_VAR

// Deterministic output projection runtime boundary.
// Single projection owner.
// No semantic/runtime authority.
// Existing global safety path preserved.

fbWaterOutputProjector(
    VI_Enable := TRUE,
    VI_System_Time_MS := GVL_STATUS.G_System_Time_MS
);

// Projection/runtime/confirmation reconciliation.
fbWaterOutputReconciliation(
    VI_Enable := TRUE,
    VI_System_Time_MS := GVL_STATUS.G_System_Time_MS
);

// Runtime bridge integrated in PRG_Water.
// This PRG remains the deterministic projection boundary.

END_PROGRAM

(* ---- PRG_Water_Output_Projection_Phase_02_Observability.st ---- *)
PROGRAM PRG_Water_Output_Projection_Phase_02_Observability
VAR
    fbPredictiveDiagnostics : FB_Predictive_Diagnostics_Runtime;
    fbForensicJournal : FB_Forensic_Journal_Runtime;
END_VAR

// Non-authoritative water runtime observability path.
// Does not write physical outputs or command shadow.

fbPredictiveDiagnostics(
    VI_Enable := TRUE,
    VI_System_Time_MS := GVL_STATUS.G_System_Time_MS
);

fbForensicJournal(
    VI_Enable := TRUE,
    VI_System_Time_MS := GVL_STATUS.G_System_Time_MS
);

// >>> BULK_SYNC_ANCHOR: PRG_Water_Output_Projection_Phase_02_Observability <<<
END_PROGRAM

(* ---- PRG_Water_Supervisory_Publication.st ---- *)
PROGRAM PRG_Water_Supervisory_Publication
VAR
    fbWaterLeakProjection : FB_Water_Leak_Runtime_Projection;
    fbWaterIsolationProjection : FB_Water_Isolation_Runtime_Projection;

    L_i : INT;
    L_State : ST_Water_Leak_Runtime_State;

    L_Any_Leak : BOOL;
    L_Any_Warning : BOOL;
    L_Any_Degraded_Mapping : BOOL;
    L_Selective_Isolation_Available : BOOL;
    L_Global_Fallback_Required : BOOL;
END_VAR

// ==============================================================================
// Water/Flood supervisory publication orchestration.
//
// Observe/publish-only.
// Does NOT mutate valve authority, runtime arbitration or safety shutdown.
// ==============================================================================

// Canonical Water semantic projection.
fbWaterLeakProjection(
    VI_Enable := TRUE,
    VI_System_Time_MS := GVL_STATUS.G_System_Time_MS
);

// Canonical Water isolation semantic projection.
fbWaterIsolationProjection(
    VI_Enable := TRUE,
    VI_System_Time_MS := GVL_STATUS.G_System_Time_MS
);

L_Any_Leak := FALSE;
L_Any_Warning := FALSE;
L_Any_Degraded_Mapping := FALSE;
L_Selective_Isolation_Available := FALSE;
L_Global_Fallback_Required := FALSE;

FOR L_i := 1 TO GVL_CONSTANTS.C_MAX_FLOOD_SENSORS DO

    L_State := GVL_Water_Runtime_Projection.G_Leak_Runtime_State[L_i];

    // Compatibility explainability mirrors.
    GVL_Water_Leak_Explainability.G_Leak_Visible[L_i] :=
        L_State.Leak_Confirmed;

    GVL_Water_Leak_Explainability.G_Warning_Visible[L_i] :=
        L_State.Leak_Warning_Active;

    GVL_Water_Leak_Explainability.G_Mapping_Valid[L_i] :=
        L_State.Mapping_Valid;

    GVL_Water_Leak_Explainability.G_Selectively_Isolatable[L_i] :=
        L_State.Selective_Isolation_Possible;

    GVL_Water_Leak_Explainability.G_Global_Fallback_Required[L_i] :=
        L_State.Fallback_Global_Isolation_Required;

    GVL_Water_Leak_Explainability.G_Leak_Confidence[L_i] :=
        L_State.Leak_Confidence;

    GVL_Water_Leak_Explainability.G_Valve_Group_Id[L_i] :=
        L_State.Valve_Group_Id;

    GVL_Water_Leak_Explainability.G_Hydraulic_Zone_Id[L_i] :=
        L_State.Hydraulic_Zone_Id;

    GVL_Water_Leak_Explainability.G_Reason_Code[L_i] :=
        L_State.Reason_Code;

    GVL_Water_Leak_Explainability.G_Reason_Text[L_i] :=
        L_State.Reason_Text;

    GVL_Water_Leak_Explainability.G_Warning_Started_Event[L_i] :=
        L_State.Warning_Started_Event;

    GVL_Water_Leak_Explainability.G_Leak_Confirmed_Event[L_i] :=
        L_State.Leak_Confirmed_Event;

    GVL_Water_Leak_Explainability.G_Leak_Cleared_Event[L_i] :=
        L_State.Leak_Cleared_Event;

    // Supervisory aggregation.
    L_Any_Leak := L_Any_Leak OR L_State.Leak_Confirmed;
    L_Any_Warning := L_Any_Warning OR L_State.Leak_Warning_Active;

    L_Any_Degraded_Mapping :=
        L_Any_Degraded_Mapping OR L_State.Mapping_Missing;

    L_Selective_Isolation_Available :=
        L_Selective_Isolation_Available
        OR L_State.Selective_Isolation_Possible;

    L_Global_Fallback_Required :=
        L_Global_Fallback_Required
        OR L_State.Fallback_Global_Isolation_Required;

    IF L_State.Leak_Confirmed THEN
        GVL_Water_Runtime_Supervisory_Publication.G_Affected_Hydraulic_Zone :=
            L_State.Hydraulic_Zone_Id;

        GVL_Water_Runtime_Supervisory_Publication.G_Affected_Valve_Group :=
            L_State.Valve_Group_Id;
    END_IF;

END_FOR;

GVL_Water_Leak_Explainability.G_Explainability_Valid := TRUE;
GVL_Water_Leak_Explainability.G_Explainability_Status_Code := 0;
GVL_Water_Leak_Explainability.G_Explainability_Status_Text :=
    'Water leak explainability publication active';

// Canonical supervisory publication.
GVL_Water_Runtime_Supervisory_Publication.G_Supervisory_Valid := TRUE;
GVL_Water_Runtime_Supervisory_Publication.G_Last_Update_MS :=
    GVL_STATUS.G_System_Time_MS;

GVL_Water_Runtime_Supervisory_Publication.G_Any_Leak_Active :=
    L_Any_Leak;

GVL_Water_Runtime_Supervisory_Publication.G_Any_Warning_Active :=
    L_Any_Warning;

GVL_Water_Runtime_Supervisory_Publication.G_Any_Degraded_Mapping :=
    L_Any_Degraded_Mapping;

GVL_Water_Runtime_Supervisory_Publication.G_Selective_Isolation_Available :=
    L_Selective_Isolation_Available;

GVL_Water_Runtime_Supervisory_Publication.G_Global_Fallback_Active :=
    L_Global_Fallback_Required;

GVL_Water_Runtime_Supervisory_Publication.G_Active_Global_Close_Path :=
    GVL_COMMAND_SHADOW.G_Close_Valve_35
    OR GVL_COMMAND_SHADOW.G_Close_Valve_36;

GVL_Water_Runtime_Supervisory_Publication.G_Active_Safety_Latch :=
    GVL_INTENT_SAFETY.I_Water_Main_Close_Required;

IF L_Global_Fallback_Required THEN
    GVL_Water_Runtime_Supervisory_Publication.G_Status_Code := 2;
    GVL_Water_Runtime_Supervisory_Publication.G_Status_Text :=
        'Global isolation fallback required';
ELSIF L_Any_Leak THEN
    GVL_Water_Runtime_Supervisory_Publication.G_Status_Code := 1;
    GVL_Water_Runtime_Supervisory_Publication.G_Status_Text :=
        'Selective isolation topology visible';
ELSIF L_Any_Warning THEN
    GVL_Water_Runtime_Supervisory_Publication.G_Status_Code := 3;
    GVL_Water_Runtime_Supervisory_Publication.G_Status_Text :=
        'Water leak warning active';
ELSE
    GVL_Water_Runtime_Supervisory_Publication.G_Status_Code := 0;
    GVL_Water_Runtime_Supervisory_Publication.G_Status_Text :=
        'Water runtime supervisory publication active';
END_IF;

// >>> BULK_SYNC_ANCHOR: PRG_Water_Supervisory_Publication <<<
END_PROGRAM

(* ---- PRG_Water_Valve_Diagnostics.st ---- *)
PROGRAM PRG_Water_Valve_Diagnostics
VAR
    L_i : INT;
    L_Now_MS : UDINT;
    L_Timeout_MS : UDINT;
    L_Elapsed_MS : UDINT;
    L_Any_Fault : BOOL;
    L_Any_Close_Fault : BOOL;
    L_First_Close_Fault : INT;
    L_Open_Command : ARRAY[1..8] OF BOOL;
    L_Close_Command : ARRAY[1..8] OF BOOL;
    L_Last_Open_Command : ARRAY[1..8] OF BOOL;
    L_Last_Close_Command : ARRAY[1..8] OF BOOL;
    L_Open_Start_MS : ARRAY[1..8] OF UDINT;
    L_Close_Start_MS : ARRAY[1..8] OF UDINT;
END_VAR

L_Now_MS := GVL_TIME_SERVICE.G_Now_MS;
L_Timeout_MS := GVL_CONSTANTS.C_MS_IN_SECOND * 10;
L_Any_Fault := FALSE;
L_Any_Close_Fault := FALSE;
L_First_Close_Fault := 0;

FOR L_i := 1 TO 6 DO
    L_Open_Command[L_i] := GVL_WATER_OUTPUT.DO_Water_Local_Valve_Open[L_i];
    L_Close_Command[L_i] := GVL_WATER_OUTPUT.DO_Water_Local_Valve_Close[L_i];
END_FOR;

L_Open_Command[7] := GVL_WATER_OUTPUT.DO_Water_Valve_35_Open;
L_Close_Command[7] := GVL_WATER_OUTPUT.DO_Water_Valve_35_Close;
L_Open_Command[8] := GVL_WATER_OUTPUT.DO_Water_Valve_36_Open;
L_Close_Command[8] := GVL_WATER_OUTPUT.DO_Water_Valve_36_Close;

FOR L_i := 1 TO 8 DO
    IF L_Open_Command[L_i] AND NOT L_Last_Open_Command[L_i] THEN
        L_Open_Start_MS[L_i] := L_Now_MS;
    END_IF;

    IF L_Close_Command[L_i] AND NOT L_Last_Close_Command[L_i] THEN
        L_Close_Start_MS[L_i] := L_Now_MS;
    END_IF;

    IF L_Open_Command[L_i] THEN
        IF GVL_STATE.G_Water_Zone_Open_FB[L_i] THEN
            GVL_STATUS.G_Diagnostics.Water_Zone_Open_Fault[L_i] := FALSE;
        ELSE
            IF L_Now_MS >= L_Open_Start_MS[L_i] THEN
                L_Elapsed_MS := L_Now_MS - L_Open_Start_MS[L_i];
            ELSE
                L_Elapsed_MS := (4294967295 - L_Open_Start_MS[L_i]) + L_Now_MS + 1;
            END_IF;
            GVL_STATUS.G_Diagnostics.Water_Zone_Open_Fault[L_i] := L_Elapsed_MS >= L_Timeout_MS;
        END_IF;
    ELSE
        GVL_STATUS.G_Diagnostics.Water_Zone_Open_Fault[L_i] := FALSE;
    END_IF;

    IF L_Close_Command[L_i] THEN
        IF GVL_STATE.G_Water_Zone_Close_FB[L_i] THEN
            GVL_STATUS.G_Diagnostics.Water_Zone_Close_Fault[L_i] := FALSE;
            GVL_STATUS.G_Diagnostics.Water_Zone_Critical_Close_Fault[L_i] := FALSE;
        ELSE
            IF L_Now_MS >= L_Close_Start_MS[L_i] THEN
                L_Elapsed_MS := L_Now_MS - L_Close_Start_MS[L_i];
            ELSE
                L_Elapsed_MS := (4294967295 - L_Close_Start_MS[L_i]) + L_Now_MS + 1;
            END_IF;
            GVL_STATUS.G_Diagnostics.Water_Zone_Close_Fault[L_i] := L_Elapsed_MS >= L_Timeout_MS;
            GVL_STATUS.G_Diagnostics.Water_Zone_Critical_Close_Fault[L_i] := L_Elapsed_MS >= L_Timeout_MS;
        END_IF;
    ELSE
        GVL_STATUS.G_Diagnostics.Water_Zone_Close_Fault[L_i] := FALSE;
        GVL_STATUS.G_Diagnostics.Water_Zone_Critical_Close_Fault[L_i] := FALSE;
    END_IF;

    IF GVL_STATUS.G_Diagnostics.Water_Zone_Open_Fault[L_i] OR GVL_STATUS.G_Diagnostics.Water_Zone_Close_Fault[L_i] THEN
        L_Any_Fault := TRUE;
    END_IF;

    IF GVL_STATUS.G_Diagnostics.Water_Zone_Critical_Close_Fault[L_i] THEN
        L_Any_Close_Fault := TRUE;
        IF L_First_Close_Fault = 0 THEN
            L_First_Close_Fault := L_i;
        END_IF;
    END_IF;

    L_Last_Open_Command[L_i] := L_Open_Command[L_i];
    L_Last_Close_Command[L_i] := L_Close_Command[L_i];
END_FOR;

GVL_STATUS.G_Diagnostics.Water_Close_Fault_Active := L_Any_Close_Fault;
GVL_STATUS.G_Diagnostics.Water_Main_Shutdown_Recommended := L_Any_Close_Fault;
GVL_STATUS.G_Diagnostics.Water_Localization_Failed := L_Any_Close_Fault;

IF L_Any_Close_Fault THEN
    GVL_STATUS.G_Diagnostics.Water_Close_Fault_Text := 'Water valve close feedback timeout';
    GVL_STATUS.G_Diagnostics.Water_Escalation_Text := 'Water close fault: common inlet fallback recommended';
    IF L_First_Close_Fault <= 6 THEN
        GVL_STATUS.G_Diagnostics.Water_Close_Fault_Zone_Name := 'Local water valve';
    ELSE
        GVL_STATUS.G_Diagnostics.Water_Close_Fault_Zone_Name := 'Common inlet valve';
    END_IF;
ELSIF NOT L_Any_Fault THEN
    GVL_STATUS.G_Diagnostics.Water_Close_Fault_Text := '';
    GVL_STATUS.G_Diagnostics.Water_Escalation_Text := '';
    GVL_STATUS.G_Diagnostics.Water_Close_Fault_Zone_Name := '';
END_IF;

// >>> BULK_SYNC_ANCHOR: PRG_Water_Valve_Diagnostics <<<
END_PROGRAM
